{attribute 'GeneratedUsingTerminal: AT2040-0250-0021'}
{attribute addProperty BoxType "AT2040-0250-0021"}
{attribute addProperty Id "A_0108_AT2000_5233_0019_AT2000_5233AT2000_01D6DEDF80"}
{attribute addProperty CRC "2568867336"}
{attribute addProperty Size "80"}
TYPE A_0036_AT2040_0250_0021_991DCE08 EXTENDS AT2040_86175B41 :
STRUCT
	{attribute addProperty Name "A_0108_AT2000_5233_0019_AT2000_5233"}
	A_0108_AT2000_5233_0019_AT2000_5233 : AT2000_01D6DEDF;
END_STRUCT
END_TYPE

(* stored: Version 1.2.0.0, ProductVersion 3.1.4024.9
   DUT A_0036_AT2040_0250_0021_991DCE08: Id {62329d77-2f8d-45fd-b1e8-aea6512e127a} *)
